// TIA Portal V19 export
VAR_GLOBAL   // PLC tag table "LB307"
   LB307_Scarico_Interno_DX_Pb_Aux_2 AT %I301.7 : Bool;   // 350SH2
   LB307_Scarico_Interno_DX_Lp_Aux_2 AT %Q301.4 : Bool;   // 350SH2
   LB307_Scarico_Interno_DX_Pb_Aux_1 AT %I301.6 : Bool;   // 350SH1
   LB307_Scarico_Interno_DX_Lp_Aux_1 AT %Q301.3 : Bool;   // 350SH1
END_VAR
